//{attribute 'qualified_only'}
//{attribute 'strict'}
TYPE E_Language :
(
	// english
	EN := 0,
	// german
	DE,
	// bulgarisch
	BG,
	
	/// zero based max language index
	eLanguage_maxIdx
);
END_TYPE

(* stored: Version 1.1.0.1
   DUT E_Language: Id {6d0788dd-5c62-4724-9f00-3f0997316c07} *)
